Universal Robots PolyScope program: CubeFinishApril2022.urp

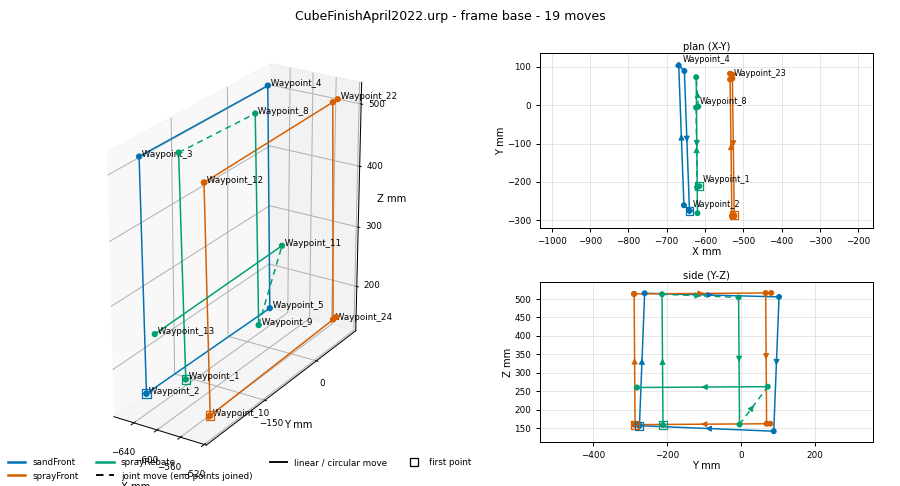
[picture p0: tool path of CubeFinishApril2022.urp in frame base, 19 of 19 moves have a stored position in this frame; points joined in program order, loops and branches not executed]
Program CubeFinishApril2022 (installation=April22Cube directory=/programs/April2022Sand/archive createdIn=5.11.5.1010327 lastSavedIn=5.11.5.1010327 robotSerialNumber=20215500677)
Calibrated DH parameters: a=[0.000204, -0.239222, -0.391845, -0.000001, 0.000022, 0]; d=[0.162722, -355.808559, 353.37206, 2.570385, 0.099741, 0.099629]; alpha=[1.571124, 0.000988, 0.008295, 1.568963, -1.570303, 0]; deltaTheta=[0, -0.973091, 7.204745, 0.05153, 0, 0]
BeforeStart
  Set DigitalOutput pin=digital_out[6]; digitalValue=0
  Call goHome
Robot Program (runOnlyOnce=false)
  Wait Sleep waitTime=0.01
  ''
  SetPayload (workpieceName=SandSpray)
SubProgram BreakEdgeFace [hidden by the author, left out]
SubProgram -> goHome
Event  expression=GoBtn ≟ True
  URCap Zero FT Sensor (Robotiq_Copilot, Robotiq Inc.) dataModel(NodeInitializedKey=true, WaitForSteadyWrenchOptionKey=true)
  Set DigitalOutput pin=ClampOn; digitalValue=1
  Call sandFront
  Call sandFront
  SuppressedNode
    MoveL speed 250 mm/s, acceleration 1200 mm/s^2 (useActiveTCP=true) feature=Base
      MoveDirectionNode (selectedDirection=ZPlus) feature(featureName=CubeFront)
        Until DISTANCE (allowActions=false deceleration=3 distanceNodeType=STOP) Distance=0.1; motionParameters(blendRadius=0)
  SuppressedNode
    Call BreakEdgeFace
  MoveL speed 250 mm/s, acceleration 1200 mm/s^2 (useActiveTCP=true) feature=Base
    MoveDirectionNode (selectedDirection=XPlus) feature(featureName=CubeFront)
      Until DISTANCE (allowActions=false deceleration=3 distanceNodeType=STOP) Distance=0.15; motionParameters(blendRadius=0)
    MoveDirectionNode (selectedDirection=ZPlus) feature(featureName=CubeFront)
      Until DISTANCE (allowActions=false deceleration=3 distanceNodeType=STOP) Distance=0.15; motionParameters(blendRadius=0)
  Call sprayFront
  Call sprayRebate
  Set DigitalOutput pin=PinsUp; digitalValue=0
  Set DigitalOutput pin=ClampOn; digitalValue=0
  Wait Sleep waitTime=1
  Call StartRotate
  Set DigitalOutput pin=ClampOn; digitalValue=1
  Call sandFront
  SuppressedNode
    MoveL speed 250 mm/s, acceleration 1200 mm/s^2 (useActiveTCP=true) feature=Base
      MoveDirectionNode (selectedDirection=ZPlus) feature(featureName=CubeFront)
        Until DISTANCE (allowActions=false deceleration=3 distanceNodeType=STOP) Distance=0.1; motionParameters(blendRadius=0)
  SuppressedNode
    Call BreakEdgeFace
  Set DigitalOutput pin=ClampOn; digitalValue=0
  MoveL speed 250 mm/s, acceleration 1200 mm/s^2 (useActiveTCP=true) feature=Base
    MoveDirectionNode (selectedDirection=ZPlus) feature(featureName=CubeFront)
      Until DISTANCE (allowActions=false deceleration=3 distanceNodeType=STOP) Distance=0.1; motionParameters(blendRadius=0)
  Call goHome
SubProgram -> sprayFront
SubProgram -> sprayRebate
Event  expression=PinsBtn≟ True
  If PinsBtn≟ True
    If PinsUp≟ True
      Set DigitalOutput pin=PinsUp; digitalValue=0
    Else 
      Set DigitalOutput pin=PinsUp; digitalValue=1
  Wait Sleep waitTime=0.5
SubProgram -> StartRotate
SubProgram -> sandFront
SubProgram goHome (keepSynchronizedWithDisk=false)
  Set SingleDigitalPulseActionState SingleDigitalPulseActionState(hiPulseInSeconds=0.1, pin=digital_out[0])
SubProgram sandFront (keepSynchronizedWithDisk=true) programFile=/programs/April2022Sand/subs/sandFront.urp
  Folder sandFront
    Set NoAction tcp=SandTCP
    MoveL speed 250 mm/s, acceleration 1200 mm/s^2 (useActiveTCP=false) tcp=SandTCP; feature=CubeFront
      Waypoint Waypoint_2: TCP in base x=-640.223 y=-275.199 z=156.226 mm, rx=-1.2204 ry=-1.2324 rz=1.2203 rad; joints [17.781, -57.17, 119.571, -107.724, 102.723, -191.638] deg; TCP offset x=3.18 y=114.64 z=98.2 mm, rx=-0.7854 ry=0 rz=0 rad; feature pose in base x=-653.492 y=-289.417 z=153.329 mm, rx=1.1922 ry=1.2015 rz=1.2274 rad
      URCap Zero FT Sensor (Robotiq_Copilot, Robotiq Inc.) dataModel(NodeInitializedKey=true, WaitForSteadyWrenchOptionKey=true)
      URCap Find Surface (Robotiq_Copilot, Robotiq Inc.) dataModel(NodeInitializedKey=true, WaitForSteadyWrenchOptionKey=false, ls_force=10.0, ls_distance=100.0, ls_speed=5.0, ZeroSensorBeforeKey=false, ls_if_distance=false, ls_if_force=false); state(isChildrenLocked=true)
        'Add Stop conditions from the Find Surface node'
      URCap Finishing Tool Control (Robotiq_Copilot, Robotiq Inc.) dataModel(ToolOutputNameKey=SanderOn, HackTriggeringContributionIsDefinedMethodKey=true)
      Wait Sleep waitTime=0.5
    MoveL speed 120 mm/s, acceleration 1200 mm/s^2 (useActiveTCP=false) tcp=SandTCP; feature=CubeFront
      Force Simple feature=Joint_6_name; selection=[0, 0, 1, 0, 0, 0]; wrench=[0, 0, 8, 0, 0, 0]; limitsForce=[0.15, 0.15, 0.15, 1.047198, 1.047198, 1.047198]; limitsMotion=[0.1, 0.1, 0.1, 0.349066, 0.349066, 0.349066]
        Waypoint Waypoint_3: TCP in base x=-654.721 y=-261.069 z=515.678 mm, rx=-1.2204 ry=-1.2324 rz=1.2203 rad; joints [15.774, -86.168, 94.118, -52.901, 101.208, -189.777] deg; TCP offset x=3.18 y=114.64 z=98.2 mm, rx=-0.7854 ry=0 rz=0 rad
        Waypoint Waypoint_4: TCP in base x=-668.238 y=103.594 z=505.785 mm, rx=-1.2204 ry=-1.2324 rz=1.2203 rad; joints [-30.039, -92.989, 103.089, -58.428, 68.843, -156.793] deg; TCP offset x=3.18 y=114.64 z=98.2 mm, rx=-0.7854 ry=0 rz=0 rad
        Waypoint Waypoint_5: TCP in base x=-653.544 y=89.234 z=141.364 mm, rx=-1.2204 ry=-1.2324 rz=1.2203 rad; joints [-29.46, -58.609, 129.969, -119.346, 69.268, -157.737] deg; TCP offset x=3.18 y=114.64 z=98.2 mm, rx=-0.7854 ry=0 rz=0 rad
        Waypoint Waypoint_6: TCP in base x=-640.229 y=-275.219 z=156.249 mm, rx=-1.2204 ry=-1.2324 rz=1.2203 rad; joints [17.783, -57.171, 119.568, -107.723, 102.726, -191.637] deg; TCP offset x=3.18 y=114.64 z=98.2 mm, rx=-0.7854 ry=0 rz=0 rad
        URCap Finishing Tool Control (Robotiq_Copilot, Robotiq Inc.) dataModel(ToolOutputNameKey=SanderOn, HackTriggeringContributionIsDefinedMethodKey=true, FinishingToolStateKey=false)
      MoveDirectionNode (selectedDirection=ZMinus) feature=Joint_6_name
        Until DISTANCE (allowActions=false deceleration=3 distanceNodeType=STOP) Distance=0.025; motionParameters(blendRadius=0)
SubProgram sprayFront (keepSynchronizedWithDisk=true) programFile=/programs/April2022Sand/subs/sprayFront.urp
  Folder SprayFront
    MoveJ speed 60 deg/s, acceleration 80 deg/s^2 (useActiveTCP=false) tcp=SprayTCP; feature=CubeFront
      Waypoint Waypoint_10: TCP in base x=-523.38 y=-287.102 z=159.121 mm, rx=2.237 ry=0.0227 rz=-2.1993 rad; joints [-1.673, -68.159, 119.265, -45.014, 43.276, 89.806] deg; TCP offset x=20.839 y=-27.14 z=105.994 mm, rx=0.1226 ry=1.1769 rz=2.8697 rad
      Set DigitalOutput pin=SprayerOn; digitalValue=1
    MoveL speed 100 mm/s, acceleration 1200 mm/s^2 (useActiveTCP=true) feature=CubeFront
      Waypoint Waypoint_12: TCP in base x=-529.431 y=-289.634 z=514.036 mm, rx=2.2371 ry=0.0226 rz=-2.1994 rad; joints [-1.244, -87.515, 84.625, 8.827, 43.306, 90.018] deg
      Set DigitalOutput pin=SprayerOn; digitalValue=0
      MoveDirectionNode (selectedDirection=ZMinus toolParams=0.2, 1.2) feature=Joint_6_name
        Until DISTANCE (allowActions=false deceleration=3 distanceNodeType=STOP) Distance=0.1; motionParameters(blendRadius=0)
    MoveJ speed 60 deg/s, acceleration 80 deg/s^2 (useActiveTCP=false) tcp=SprayTCP; feature=CubeFront
      Waypoint Waypoint_21: TCP in base x=-529.452 y=-289.651 z=513.978 mm, rx=1.2334 ry=-1.2087 rz=-1.1964 rad; joints [21.172, -83.163, 107.28, -68.757, 101.457, 169.304] deg
      Set DigitalOutput pin=SprayerOn; digitalValue=1
    MoveL speed 100 mm/s, acceleration 1200 mm/s^2 (useActiveTCP=false) tcp=SprayTCP; feature=CubeFront
      Waypoint Waypoint_22: TCP in base x=-534.417 y=82.311 z=516.561 mm, rx=1.2336 ry=-1.2085 rz=-1.1962 rad; joints [-29.561, -95.964, 120.769, -74.274, 65.61, 206.091] deg
      Set DigitalOutput pin=SprayerOn; digitalValue=0
      MoveDirectionNode (selectedDirection=ZMinus toolParams=0.2, 1.2) feature=Joint_6_name
        Until DISTANCE (allowActions=false deceleration=3 distanceNodeType=STOP) Distance=0.1; motionParameters(blendRadius=0)
    MoveJ speed 60 deg/s, acceleration 80 deg/s^2 (useActiveTCP=false) tcp=SprayTCP; feature=CubeFront
      Waypoint Waypoint_23: TCP in base x=-534.231 y=67.346 z=516.387 mm, rx=0.0162 ry=-1.5879 rz=0.0049 rad; joints [-5.513, -90.525, 84.578, 2.415, 128.236, 270.805] deg
      Set DigitalOutput pin=SprayerOn; digitalValue=1
    MoveL speed 100 mm/s, acceleration 1200 mm/s^2 (useActiveTCP=false) tcp=SprayTCP; feature=CubeFront
      Waypoint Waypoint_24: TCP in base x=-528.185 y=69.879 z=161.61 mm, rx=0.0161 ry=-1.5879 rz=0.005 rad; joints [-6.031, -73.189, 122.225, -52.664, 128.115, 270.655] deg
      Set DigitalOutput pin=SprayerOn; digitalValue=0
      MoveDirectionNode (selectedDirection=ZMinus toolParams=0.2, 1.2) feature=Joint_6_name
        Until DISTANCE (allowActions=false deceleration=3 distanceNodeType=STOP) Distance=0.1; motionParameters(blendRadius=0)
    MoveJ speed 60 deg/s, acceleration 80 deg/s^2 (useActiveTCP=false) tcp=SprayTCP; feature=CubeFront
      Waypoint Waypoint_38: TCP in base x=-528.29 y=79.87 z=161.661 mm, rx=1.2332 ry=-1.2085 rz=-1.1965 rad; joints [-29.8, -43.92, 133.995, -139.433, 65.363, 205.789] deg
      Set DigitalOutput pin=SprayerOn; digitalValue=1
    MoveL speed 100 mm/s, acceleration 1200 mm/s^2 (useActiveTCP=false) tcp=SprayTCP; feature=CubeFront
      Waypoint Waypoint_25: TCP in base x=-523.325 y=-290.033 z=159.067 mm, rx=1.2331 ry=-1.2086 rz=-1.1966 rad; joints [21.408, -42.582, 119.14, -121.322, 101.623, 168.739] deg
      Set DigitalOutput pin=SprayerOn; digitalValue=0
      MoveDirectionNode (selectedDirection=ZMinus toolParams=0.2, 1.2) feature=Joint_6_name
        Until DISTANCE (allowActions=false deceleration=3 distanceNodeType=STOP) Distance=0.1; motionParameters(blendRadius=0)
SubProgram sprayRebate (keepSynchronizedWithDisk=true) programFile=/programs/April2022Sand/subs/sprayRebate.urp
  Folder SprayRebate
    MoveJ speed 60 deg/s, acceleration 80 deg/s^2 (useActiveTCP=false) tcp=SprayTCP; feature=CubeFront
      Waypoint Waypoint_1: TCP in base x=-614.395 y=-211.304 z=158.056 mm, rx=0.8919 ry=-1.3989 rz=0.8972 rad; joints [3.832, -69.113, 116.159, -49.553, 73.09, -85.388] deg
      Set DigitalOutput pin=SprayerOn; digitalValue=1
    MoveL speed 100 mm/s, acceleration 1200 mm/s^2 (useActiveTCP=true) feature=CubeFront
      Waypoint Waypoint_7: TCP in base x=-620.397 y=-213.913 z=513.046 mm, rx=0.892 ry=-1.3988 rz=0.8971 rad; joints [4.169, -85.315, 79.236, 3.53, 73.033, -85.264] deg
      Set DigitalOutput pin=SprayerOn; digitalValue=0
      MoveDirectionNode (selectedDirection=ZPlus toolParams=0.2, 1.2)
        Until DISTANCE (allowActions=false deceleration=3 distanceNodeType=STOP) Distance=0.1; motionParameters(blendRadius=0)
    MoveJ speed 60 deg/s, acceleration 80 deg/s^2 (useActiveTCP=false) tcp=SprayTCP; feature=CubeFront
      Waypoint Waypoint_8: TCP in base x=-623.058 y=-6.085 z=504.453 mm, rx=-1.5379 ry=0.9456 rz=1.5188 rad; joints [-11.433, -87.799, 86.311, 5.702, 98.013, 93.92] deg
      Set DigitalOutput pin=SprayerOn; digitalValue=1
    MoveL speed 100 mm/s, acceleration 1200 mm/s^2 (useActiveTCP=false) tcp=SprayTCP; feature=CubeFront
      Waypoint Waypoint_9: TCP in base x=-617.186 y=-3.636 z=159.537 mm, rx=-1.538 ry=0.9455 rz=1.5188 rad; joints [-11.994, -68.384, 119.511, -46.936, 97.835, 93.758] deg
      Set DigitalOutput pin=SprayerOn; digitalValue=0
      MoveDirectionNode (selectedDirection=ZPlus toolParams=0.2, 1.2)
        Until DISTANCE (allowActions=false deceleration=3 distanceNodeType=STOP) Distance=0.1; motionParameters(blendRadius=0)
    MoveJ speed 60 deg/s, acceleration 80 deg/s^2 (useActiveTCP=false) tcp=SprayTCP; feature=CubeFront
      Waypoint Waypoint_11: TCP in base x=-622.643 y=73.149 z=262.251 mm, rx=2.0067 ry=-1.985 rz=-0.4223 rad; joints [-27.089, -68.36, 126.552, 146.432, -61.498, -7.368] deg; TCP offset x=20.839 y=-27.14 z=105.994 mm, rx=0.1226 ry=1.1769 rz=2.8697 rad
      Set DigitalOutput pin=SprayerOn; digitalValue=1
    MoveL speed 100 mm/s, acceleration 1200 mm/s^2 (useActiveTCP=false) tcp=SprayTCP; feature=CubeFront
      Waypoint Waypoint_13: TCP in base x=-619.354 y=-281.828 z=259.921 mm, rx=2.0066 ry=-1.9851 rz=-0.4224 rad; joints [19.517, -59.938, 112.11, 150.357, -104.552, 371.006] deg; TCP offset x=20.839 y=-27.14 z=105.994 mm, rx=0.1226 ry=1.1769 rz=2.8697 rad
      Set DigitalOutput pin=SprayerOn; digitalValue=0
      MoveDirectionNode (selectedDirection=ZPlus toolParams=0.2, 1.2)
        Until DISTANCE (allowActions=false deceleration=3 distanceNodeType=STOP) Distance=0.1; motionParameters(blendRadius=0)
SubProgram StartRotate (keepSynchronizedWithDisk=false)
  Set AnalogOutput pin=RotateGo; analogValue=4
  Wait Sleep waitTime=0.1
  Set AnalogOutput pin=RotateGo; analogValue=0
  Wait Sleep waitTime=10
